Fanuc KAREL source: kt00030.KL

-- PROVISIONAL review KL for V1013-1; original PC SHA256 6f6fbf8945775663fd585379e71be4bebef76d4bf3b7fe6ccfd954edc8307312
-- Incomplete behavior may be omitted. Consult companion uncertainty JSON. Do not deploy.
PROGRAM KT00030
%NOLOCKGROUP
VAR
  OUT : REAL
-- UNRESOLVED_DECL H1 type=002017
-- UNRESOLVED_DECL Y2 type=002018
BEGIN
  -- UNRESOLVED_PC offsets 5-19; opcodes 2E,22,9D,33,B4
  -- UNRESOLVED_PC offsets 24-38; opcodes 2E,22,9D,33,B2
  -- UNRESOLVED_PC offsets 43-69; opcodes 22,9D,33,B3,22,9D,33,B1,52,64,23
  -- UNRESOLVED_PC offsets 74-78; opcodes 7F
END KT00030
